REGION Network 42: Assign PLC Alarm Text List
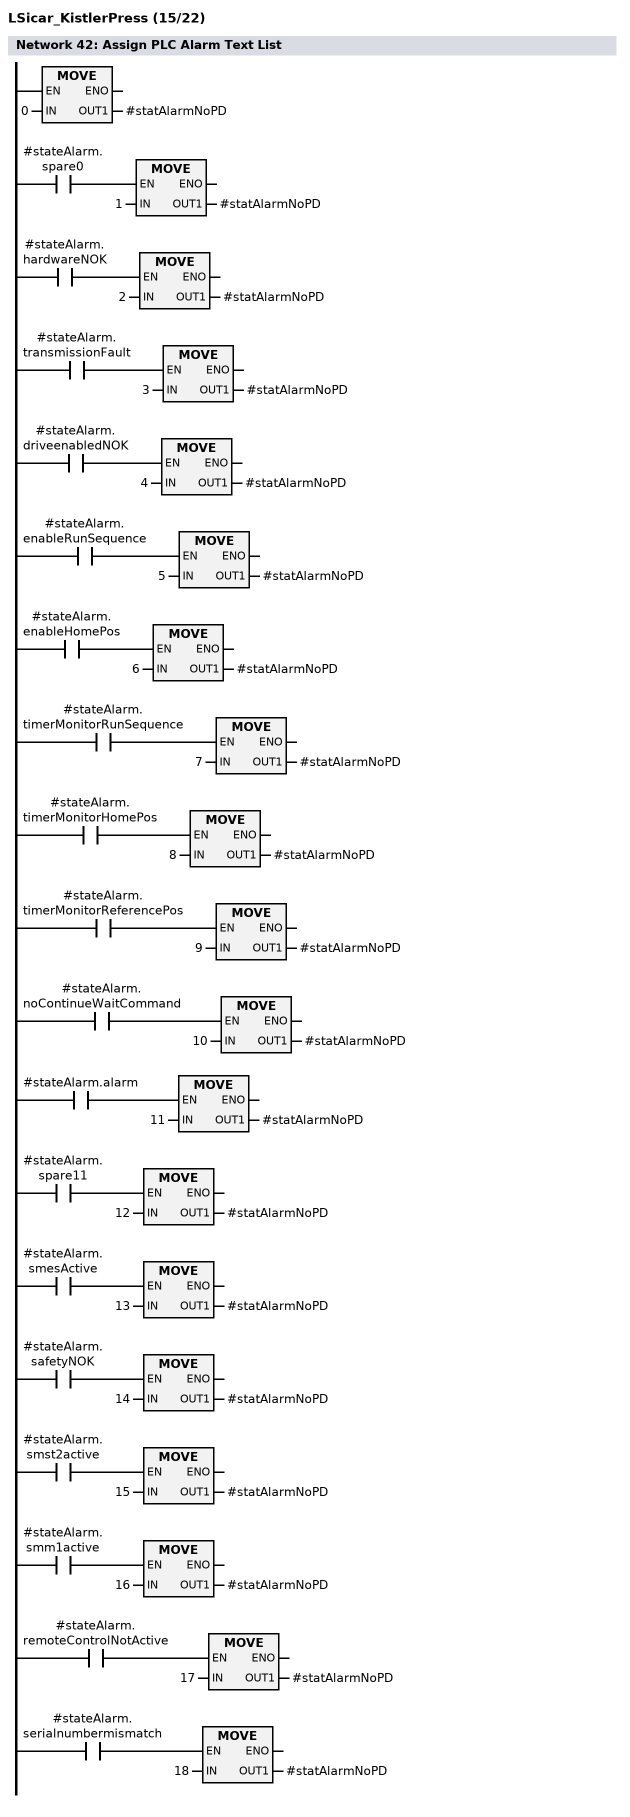
   RUNG wire#powerrail
      Move(in := 0, out1 => #statAlarmNoPD)
   END_RUNG
   RUNG wire#powerrail
      Contact( #stateAlarm.spare0 )
      Move(in := 1, out1 => #statAlarmNoPD)
   END_RUNG
   RUNG wire#powerrail
      Contact( #stateAlarm.hardwareNOK )
      Move(in := 2, out1 => #statAlarmNoPD)
   END_RUNG
   RUNG wire#powerrail
      Contact( #stateAlarm.transmissionFault )
      Move(in := 3, out1 => #statAlarmNoPD)
   END_RUNG
   RUNG wire#powerrail
      Contact( #stateAlarm.driveenabledNOK )
      Move(in := 4, out1 => #statAlarmNoPD)
   END_RUNG
   RUNG wire#powerrail
      Contact( #stateAlarm.enableRunSequence )
      Move(in := 5, out1 => #statAlarmNoPD)
   END_RUNG
   RUNG wire#powerrail
      Contact( #stateAlarm.enableHomePos )
      Move(in := 6, out1 => #statAlarmNoPD)
   END_RUNG
   RUNG wire#powerrail
      Contact( #stateAlarm.timerMonitorRunSequence )
      Move(in := 7, out1 => #statAlarmNoPD)
   END_RUNG
   RUNG wire#powerrail
      Contact( #stateAlarm.timerMonitorHomePos )
      Move(in := 8, out1 => #statAlarmNoPD)
   END_RUNG
   RUNG wire#powerrail
      Contact( #stateAlarm.timerMonitorReferencePos )
      Move(in := 9, out1 => #statAlarmNoPD)
   END_RUNG
   RUNG wire#powerrail
      Contact( #stateAlarm.noContinueWaitCommand )
      Move(in := 10, out1 => #statAlarmNoPD)
   END_RUNG
   RUNG wire#powerrail
      Contact( #stateAlarm.alarm )
      Move(in := 11, out1 => #statAlarmNoPD)
   END_RUNG
   RUNG wire#powerrail
      Contact( #stateAlarm.spare11 )
      Move(in := 12, out1 => #statAlarmNoPD)
   END_RUNG
   RUNG wire#powerrail
      Contact( #stateAlarm.smesActive )
      Move(in := 13, out1 => #statAlarmNoPD)
   END_RUNG
   RUNG wire#powerrail
      Contact( #stateAlarm.safetyNOK )
      Move(in := 14, out1 => #statAlarmNoPD)
   END_RUNG
   RUNG wire#powerrail
      Contact( #stateAlarm.smst2active )
      Move(in := 15, out1 => #statAlarmNoPD)
   END_RUNG
   RUNG wire#powerrail
      Contact( #stateAlarm.smm1active )
      Move(in := 16, out1 => #statAlarmNoPD)
   END_RUNG
   RUNG wire#powerrail
      Contact( #stateAlarm.remoteControlNotActive )
      Move(in := 17, out1 => #statAlarmNoPD)
   END_RUNG
   RUNG wire#powerrail
      Contact( #stateAlarm.serialnumbermismatch )
      Move(in := 18, out1 => #statAlarmNoPD)
   END_RUNG
   // the same network as SCL:
   #statAlarmNoPD := 0;
   IF #stateAlarm.spare0 THEN #statAlarmNoPD := 1; END_IF;
   IF #stateAlarm.hardwareNOK THEN #statAlarmNoPD := 2; END_IF;
   IF #stateAlarm.transmissionFault THEN #statAlarmNoPD := 3; END_IF;
   IF #stateAlarm.driveenabledNOK THEN #statAlarmNoPD := 4; END_IF;
   IF #stateAlarm.enableRunSequence THEN #statAlarmNoPD := 5; END_IF;
   IF #stateAlarm.enableHomePos THEN #statAlarmNoPD := 6; END_IF;
   IF #stateAlarm.timerMonitorRunSequence THEN #statAlarmNoPD := 7; END_IF;
   IF #stateAlarm.timerMonitorHomePos THEN #statAlarmNoPD := 8; END_IF;
   IF #stateAlarm.timerMonitorReferencePos THEN #statAlarmNoPD := 9; END_IF;
   IF #stateAlarm.noContinueWaitCommand THEN #statAlarmNoPD := 10; END_IF;
   IF #stateAlarm.alarm THEN #statAlarmNoPD := 11; END_IF;
   IF #stateAlarm.spare11 THEN #statAlarmNoPD := 12; END_IF;
   IF #stateAlarm.smesActive THEN #statAlarmNoPD := 13; END_IF;
   IF #stateAlarm.safetyNOK THEN #statAlarmNoPD := 14; END_IF;
   IF #stateAlarm.smst2active THEN #statAlarmNoPD := 15; END_IF;
   IF #stateAlarm.smm1active THEN #statAlarmNoPD := 16; END_IF;
   IF #stateAlarm.remoteControlNotActive THEN #statAlarmNoPD := 17; END_IF;
   IF #stateAlarm.serialnumbermismatch THEN #statAlarmNoPD := 18; END_IF;
END_REGION

REGION Network 43: HMI Color Association
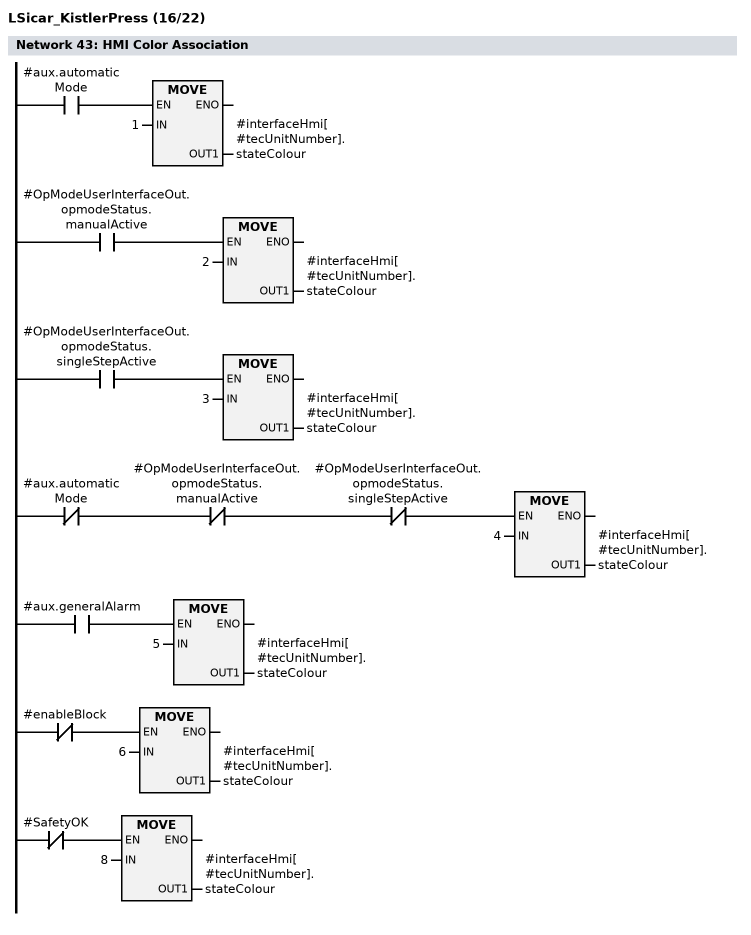
   RUNG wire#powerrail
      Contact( #aux.automaticMode )
      Move(in := 1, out1 => #interfaceHmi[#tecUnitNumber].stateColour)
   END_RUNG
   RUNG wire#powerrail
      Contact( #OpModeUserInterfaceOut.opmodeStatus.manualActive )
      Move(in := 2, out1 => #interfaceHmi[#tecUnitNumber].stateColour)
   END_RUNG
   RUNG wire#powerrail
      Contact( #OpModeUserInterfaceOut.opmodeStatus.singleStepActive )
      Move(in := 3, out1 => #interfaceHmi[#tecUnitNumber].stateColour)
   END_RUNG
   RUNG wire#powerrail
      I_Contact( #aux.automaticMode )
      I_Contact( #OpModeUserInterfaceOut.opmodeStatus.manualActive )
      I_Contact( #OpModeUserInterfaceOut.opmodeStatus.singleStepActive )
      Move(in := 4, out1 => #interfaceHmi[#tecUnitNumber].stateColour)
   END_RUNG
   RUNG wire#powerrail
      Contact( #aux.generalAlarm )
      Move(in := 5, out1 => #interfaceHmi[#tecUnitNumber].stateColour)
   END_RUNG
   RUNG wire#powerrail
      I_Contact( #enableBlock )
      Move(in := 6, out1 => #interfaceHmi[#tecUnitNumber].stateColour)
   END_RUNG
   RUNG wire#powerrail
      I_Contact( #SafetyOK )
      Move(in := 8, out1 => #interfaceHmi[#tecUnitNumber].stateColour)
   END_RUNG
   // the same network as SCL:
   IF #aux.automaticMode THEN #interfaceHmi[#tecUnitNumber].stateColour := 1; END_IF;
   IF #OpModeUserInterfaceOut.opmodeStatus.manualActive THEN
       #interfaceHmi[#tecUnitNumber].stateColour := 2;
   END_IF;
   IF #OpModeUserInterfaceOut.opmodeStatus.singleStepActive THEN
       #interfaceHmi[#tecUnitNumber].stateColour := 3;
   END_IF;
   IF NOT #aux.automaticMode AND NOT #OpModeUserInterfaceOut.opmodeStatus.manualActive AND NOT #OpModeUserInterfaceOut.opmodeStatus.singleStepActive THEN
       #interfaceHmi[#tecUnitNumber].stateColour := 4;
   END_IF;
   IF #aux.generalAlarm THEN #interfaceHmi[#tecUnitNumber].stateColour := 5; END_IF;
   IF NOT #enableBlock THEN #interfaceHmi[#tecUnitNumber].stateColour := 6; END_IF;
   IF NOT #SafetyOK THEN #interfaceHmi[#tecUnitNumber].stateColour := 8; END_IF;
END_REGION

REGION Network 44: HMI state Mapping
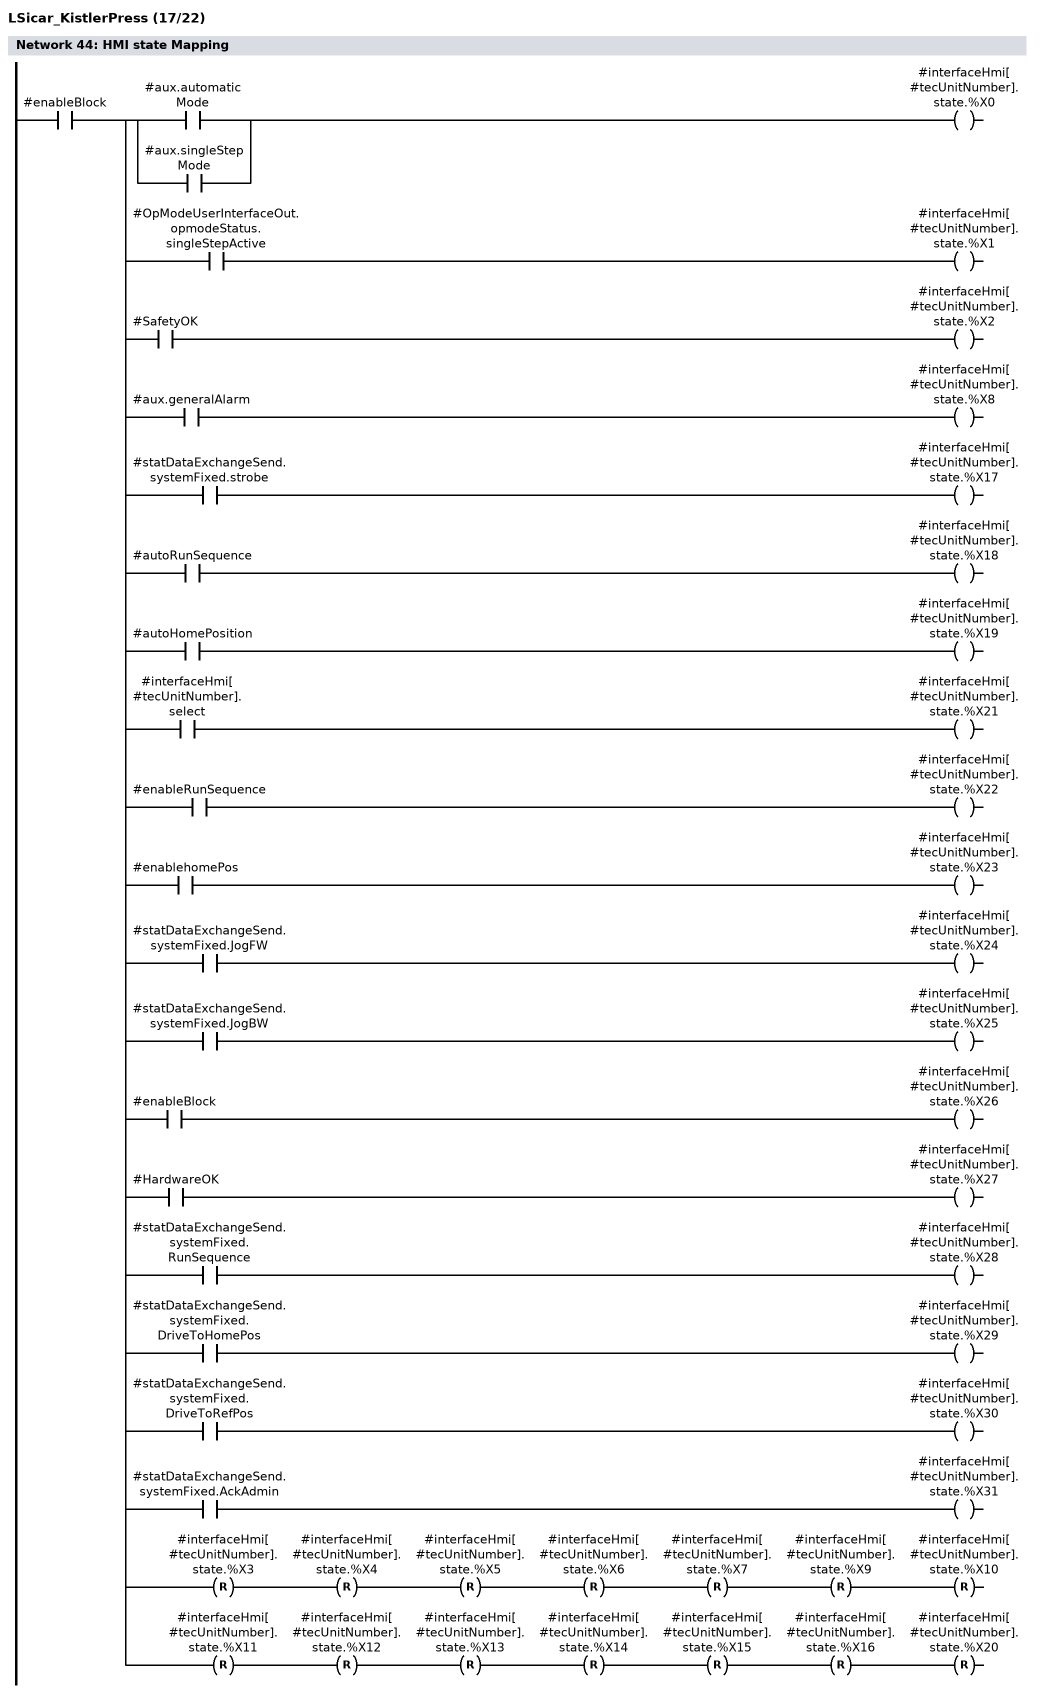
   RUNG wire#powerrail
      Contact( #enableBlock )
      wire#w1
      Contact( #aux.automaticMode )
      wire#w2
      Coil( #interfaceHmi[#tecUnitNumber].state.%X0 )
   END_RUNG
   RUNG wire#w1
      Contact( #aux.singleStepMode )
   END_RUNG wire#w2
   RUNG wire#w1
      Contact( #OpModeUserInterfaceOut.opmodeStatus.singleStepActive )
      Coil( #interfaceHmi[#tecUnitNumber].state.%X1 )
   END_RUNG
   RUNG wire#w1
      Contact( #SafetyOK )
      Coil( #interfaceHmi[#tecUnitNumber].state.%X2 )
   END_RUNG
   RUNG wire#w1
      Contact( #aux.generalAlarm )
      Coil( #interfaceHmi[#tecUnitNumber].state.%X8 )
   END_RUNG
   RUNG wire#w1
      Contact( #statDataExchangeSend.systemFixed.strobe )
      Coil( #interfaceHmi[#tecUnitNumber].state.%X17 )
   END_RUNG
   RUNG wire#w1
      Contact( #autoRunSequence )
      Coil( #interfaceHmi[#tecUnitNumber].state.%X18 )
   END_RUNG
   RUNG wire#w1
      Contact( #autoHomePosition )
      Coil( #interfaceHmi[#tecUnitNumber].state.%X19 )
   END_RUNG
   RUNG wire#w1
      Contact( #interfaceHmi[#tecUnitNumber].select )
      Coil( #interfaceHmi[#tecUnitNumber].state.%X21 )
   END_RUNG
   RUNG wire#w1
      Contact( #enableRunSequence )
      Coil( #interfaceHmi[#tecUnitNumber].state.%X22 )
   END_RUNG
   RUNG wire#w1
      Contact( #enablehomePos )
      Coil( #interfaceHmi[#tecUnitNumber].state.%X23 )
   END_RUNG
   RUNG wire#w1
      Contact( #statDataExchangeSend.systemFixed.JogFW )
      Coil( #interfaceHmi[#tecUnitNumber].state.%X24 )
   END_RUNG
   RUNG wire#w1
      Contact( #statDataExchangeSend.systemFixed.JogBW )
      Coil( #interfaceHmi[#tecUnitNumber].state.%X25 )
   END_RUNG
   RUNG wire#w1
      Contact( #enableBlock )
      Coil( #interfaceHmi[#tecUnitNumber].state.%X26 )
   END_RUNG
   RUNG wire#w1
      Contact( #HardwareOK )
      Coil( #interfaceHmi[#tecUnitNumber].state.%X27 )
   END_RUNG
   RUNG wire#w1
      Contact( #statDataExchangeSend.systemFixed.RunSequence )
      Coil( #interfaceHmi[#tecUnitNumber].state.%X28 )
   END_RUNG
   RUNG wire#w1
      Contact( #statDataExchangeSend.systemFixed.DriveToHomePos )
      Coil( #interfaceHmi[#tecUnitNumber].state.%X29 )
   END_RUNG
   RUNG wire#w1
      Contact( #statDataExchangeSend.systemFixed.DriveToRefPos )
      Coil( #interfaceHmi[#tecUnitNumber].state.%X30 )
   END_RUNG
   RUNG wire#w1
      Contact( #statDataExchangeSend.systemFixed.AckAdmin )
      Coil( #interfaceHmi[#tecUnitNumber].state.%X31 )
   END_RUNG
   RUNG wire#w1
      R_Coil( #interfaceHmi[#tecUnitNumber].state.%X3 )
      R_Coil( #interfaceHmi[#tecUnitNumber].state.%X4 )
      R_Coil( #interfaceHmi[#tecUnitNumber].state.%X5 )
      R_Coil( #interfaceHmi[#tecUnitNumber].state.%X6 )
      R_Coil( #interfaceHmi[#tecUnitNumber].state.%X7 )
      R_Coil( #interfaceHmi[#tecUnitNumber].state.%X9 )
      R_Coil( #interfaceHmi[#tecUnitNumber].state.%X10 )
   END_RUNG
   RUNG wire#w1
      R_Coil( #interfaceHmi[#tecUnitNumber].state.%X11 )
      R_Coil( #interfaceHmi[#tecUnitNumber].state.%X12 )
      R_Coil( #interfaceHmi[#tecUnitNumber].state.%X13 )
      R_Coil( #interfaceHmi[#tecUnitNumber].state.%X14 )
      R_Coil( #interfaceHmi[#tecUnitNumber].state.%X15 )
      R_Coil( #interfaceHmi[#tecUnitNumber].state.%X16 )
      R_Coil( #interfaceHmi[#tecUnitNumber].state.%X20 )
   END_RUNG
   // the same network as SCL:
   #interfaceHmi[#tecUnitNumber].state.%X0 := #enableBlock AND (#aux.automaticMode OR #aux.singleStepMode);
   #interfaceHmi[#tecUnitNumber].state.%X1 := #enableBlock AND #OpModeUserInterfaceOut.opmodeStatus.singleStepActive;
   #interfaceHmi[#tecUnitNumber].state.%X2 := #enableBlock AND #SafetyOK;
   #interfaceHmi[#tecUnitNumber].state.%X8 := #enableBlock AND #aux.generalAlarm;
   #interfaceHmi[#tecUnitNumber].state.%X17 := #enableBlock AND #statDataExchangeSend.systemFixed.strobe;
   #interfaceHmi[#tecUnitNumber].state.%X18 := #enableBlock AND #autoRunSequence;
   #interfaceHmi[#tecUnitNumber].state.%X19 := #enableBlock AND #autoHomePosition;
   #interfaceHmi[#tecUnitNumber].state.%X21 := #enableBlock AND #interfaceHmi[#tecUnitNumber].select;
   #interfaceHmi[#tecUnitNumber].state.%X22 := #enableBlock AND #enableRunSequence;
   #interfaceHmi[#tecUnitNumber].state.%X23 := #enableBlock AND #enablehomePos;
   #interfaceHmi[#tecUnitNumber].state.%X24 := #enableBlock AND #statDataExchangeSend.systemFixed.JogFW;
   #interfaceHmi[#tecUnitNumber].state.%X25 := #enableBlock AND #statDataExchangeSend.systemFixed.JogBW;
   #interfaceHmi[#tecUnitNumber].state.%X26 := #enableBlock AND #enableBlock;
   #interfaceHmi[#tecUnitNumber].state.%X27 := #enableBlock AND #HardwareOK;
   #interfaceHmi[#tecUnitNumber].state.%X28 := #enableBlock AND #statDataExchangeSend.systemFixed.RunSequence;
   #interfaceHmi[#tecUnitNumber].state.%X29 := #enableBlock AND #statDataExchangeSend.systemFixed.DriveToHomePos;
   #interfaceHmi[#tecUnitNumber].state.%X30 := #enableBlock AND #statDataExchangeSend.systemFixed.DriveToRefPos;
   #interfaceHmi[#tecUnitNumber].state.%X31 := #enableBlock AND #statDataExchangeSend.systemFixed.AckAdmin;
   IF #enableBlock THEN
       #interfaceHmi[#tecUnitNumber].state.%X3 := FALSE;
       #interfaceHmi[#tecUnitNumber].state.%X4 := FALSE;
       #interfaceHmi[#tecUnitNumber].state.%X5 := FALSE;
       #interfaceHmi[#tecUnitNumber].state.%X6 := FALSE;
       #interfaceHmi[#tecUnitNumber].state.%X7 := FALSE;
       #interfaceHmi[#tecUnitNumber].state.%X9 := FALSE;
       #interfaceHmi[#tecUnitNumber].state.%X10 := FALSE;
       #interfaceHmi[#tecUnitNumber].state.%X11 := FALSE;
       #interfaceHmi[#tecUnitNumber].state.%X12 := FALSE;
       #interfaceHmi[#tecUnitNumber].state.%X13 := FALSE;
       #interfaceHmi[#tecUnitNumber].state.%X14 := FALSE;
       #interfaceHmi[#tecUnitNumber].state.%X15 := FALSE;
       #interfaceHmi[#tecUnitNumber].state.%X16 := FALSE;
       #interfaceHmi[#tecUnitNumber].state.%X20 := FALSE;
   END_IF;
END_REGION

REGION Network 45: Send Process Values to HMI
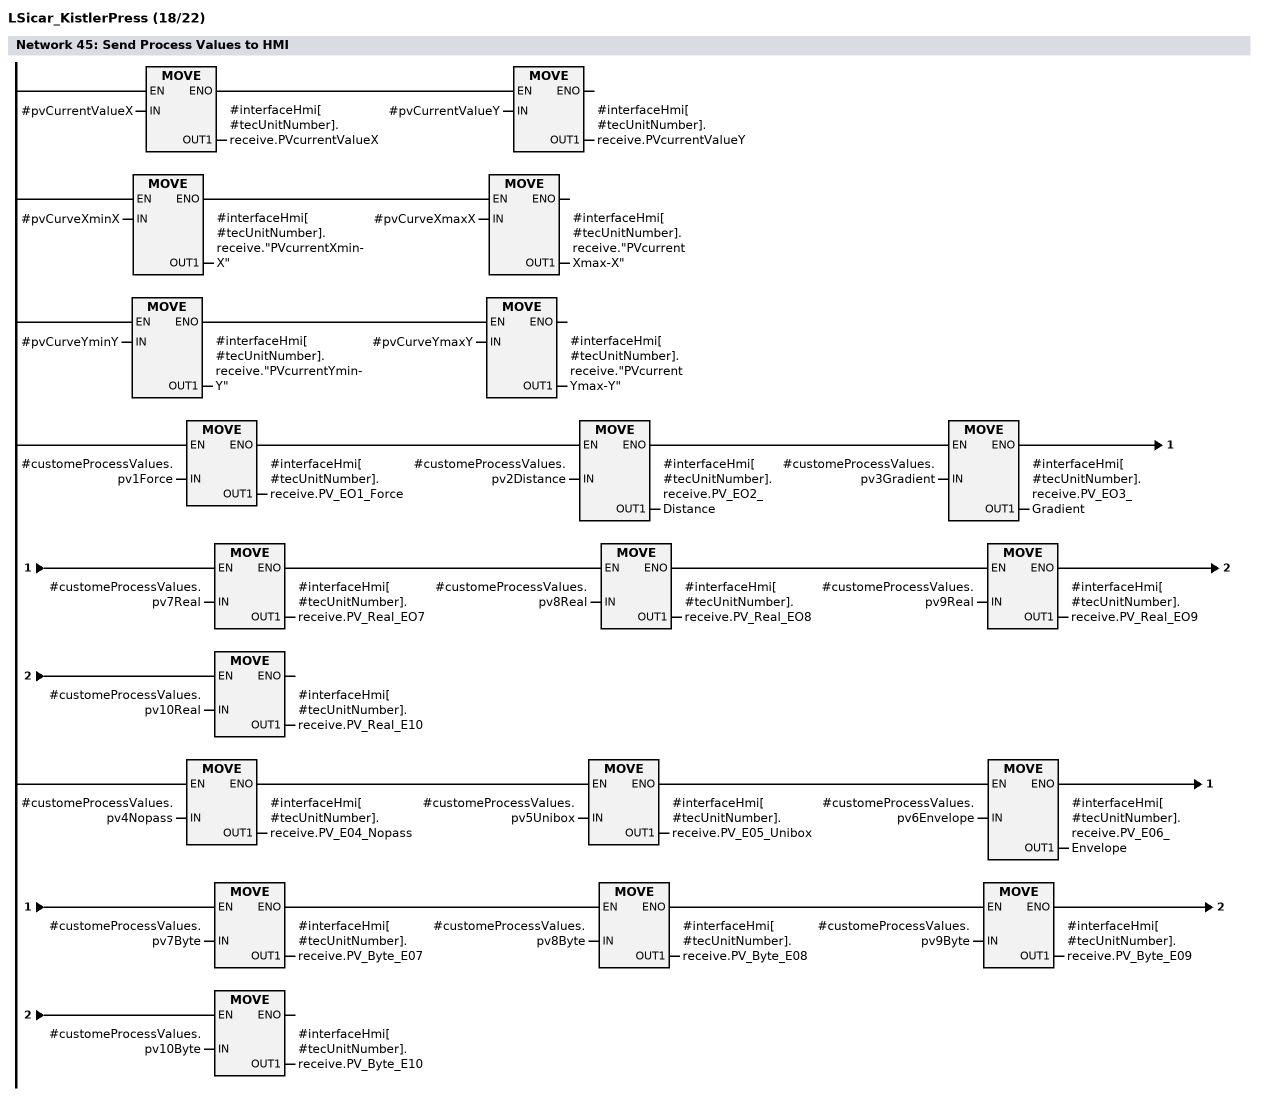
   RUNG wire#powerrail
      Move(in := #pvCurrentValueX, out1 => #interfaceHmi[#tecUnitNumber].receive.PVcurrentValueX)
      Move(in := #pvCurrentValueY, out1 => #interfaceHmi[#tecUnitNumber].receive.PVcurrentValueY)
   END_RUNG
   RUNG wire#powerrail
      Move(in := #pvCurveXminX, out1 => #interfaceHmi[#tecUnitNumber].receive."PVcurrentXmin-X")
      Move(in := #pvCurveXmaxX, out1 => #interfaceHmi[#tecUnitNumber].receive."PVcurrentXmax-X")
   END_RUNG
   RUNG wire#powerrail
      Move(in := #pvCurveYminY, out1 => #interfaceHmi[#tecUnitNumber].receive."PVcurrentYmin-Y")
      Move(in := #pvCurveYmaxY, out1 => #interfaceHmi[#tecUnitNumber].receive."PVcurrentYmax-Y")
   END_RUNG
   RUNG wire#powerrail
      Move(in := #customeProcessValues.pv1Force, out1 => #interfaceHmi[#tecUnitNumber].receive.PV_EO1_Force)
      Move(in := #customeProcessValues.pv2Distance, out1 => #interfaceHmi[#tecUnitNumber].receive.PV_EO2_Distance)
      Move(in := #customeProcessValues.pv3Gradient, out1 => #interfaceHmi[#tecUnitNumber].receive.PV_EO3_Gradient)
      Move(in := #customeProcessValues.pv7Real, out1 => #interfaceHmi[#tecUnitNumber].receive.PV_Real_EO7)
      Move(in := #customeProcessValues.pv8Real, out1 => #interfaceHmi[#tecUnitNumber].receive.PV_Real_EO8)
      Move(in := #customeProcessValues.pv9Real, out1 => #interfaceHmi[#tecUnitNumber].receive.PV_Real_EO9)
      Move(in := #customeProcessValues.pv10Real, out1 => #interfaceHmi[#tecUnitNumber].receive.PV_Real_E10)
   END_RUNG
   RUNG wire#powerrail
      Move(in := #customeProcessValues.pv4Nopass, out1 => #interfaceHmi[#tecUnitNumber].receive.PV_E04_Nopass)
      Move(in := #customeProcessValues.pv5Unibox, out1 => #interfaceHmi[#tecUnitNumber].receive.PV_E05_Unibox)
      Move(in := #customeProcessValues.pv6Envelope, out1 => #interfaceHmi[#tecUnitNumber].receive.PV_E06_Envelope)
      Move(in := #customeProcessValues.pv7Byte, out1 => #interfaceHmi[#tecUnitNumber].receive.PV_Byte_E07)
      Move(in := #customeProcessValues.pv8Byte, out1 => #interfaceHmi[#tecUnitNumber].receive.PV_Byte_E08)
      Move(in := #customeProcessValues.pv9Byte, out1 => #interfaceHmi[#tecUnitNumber].receive.PV_Byte_E09)
      Move(in := #customeProcessValues.pv10Byte, out1 => #interfaceHmi[#tecUnitNumber].receive.PV_Byte_E10)
   END_RUNG
   // the same network as SCL:
   #interfaceHmi[#tecUnitNumber].receive.PVcurrentValueX := #pvCurrentValueX;
   #interfaceHmi[#tecUnitNumber].receive.PVcurrentValueY := #pvCurrentValueY;
   #interfaceHmi[#tecUnitNumber].receive."PVcurrentXmin-X" := #pvCurveXminX;
   #interfaceHmi[#tecUnitNumber].receive."PVcurrentXmax-X" := #pvCurveXmaxX;
   #interfaceHmi[#tecUnitNumber].receive."PVcurrentYmin-Y" := #pvCurveYminY;
   #interfaceHmi[#tecUnitNumber].receive."PVcurrentYmax-Y" := #pvCurveYmaxY;
   #interfaceHmi[#tecUnitNumber].receive.PV_EO1_Force := #customeProcessValues.pv1Force;
   #interfaceHmi[#tecUnitNumber].receive.PV_EO2_Distance := #customeProcessValues.pv2Distance;
   #interfaceHmi[#tecUnitNumber].receive.PV_EO3_Gradient := #customeProcessValues.pv3Gradient;
   #interfaceHmi[#tecUnitNumber].receive.PV_Real_EO7 := #customeProcessValues.pv7Real;
   #interfaceHmi[#tecUnitNumber].receive.PV_Real_EO8 := #customeProcessValues.pv8Real;
   #interfaceHmi[#tecUnitNumber].receive.PV_Real_EO9 := #customeProcessValues.pv9Real;
   #interfaceHmi[#tecUnitNumber].receive.PV_Real_E10 := #customeProcessValues.pv10Real;
   #interfaceHmi[#tecUnitNumber].receive.PV_E04_Nopass := #customeProcessValues.pv4Nopass;
   #interfaceHmi[#tecUnitNumber].receive.PV_E05_Unibox := #customeProcessValues.pv5Unibox;
   #interfaceHmi[#tecUnitNumber].receive.PV_E06_Envelope := #customeProcessValues.pv6Envelope;
   #interfaceHmi[#tecUnitNumber].receive.PV_Byte_E07 := #customeProcessValues.pv7Byte;
   #interfaceHmi[#tecUnitNumber].receive.PV_Byte_E08 := #customeProcessValues.pv8Byte;
   #interfaceHmi[#tecUnitNumber].receive.PV_Byte_E09 := #customeProcessValues.pv9Byte;
   #interfaceHmi[#tecUnitNumber].receive.PV_Byte_E10 := #customeProcessValues.pv10Byte;
END_REGION

REGION Network 46: Enable HMI Code View
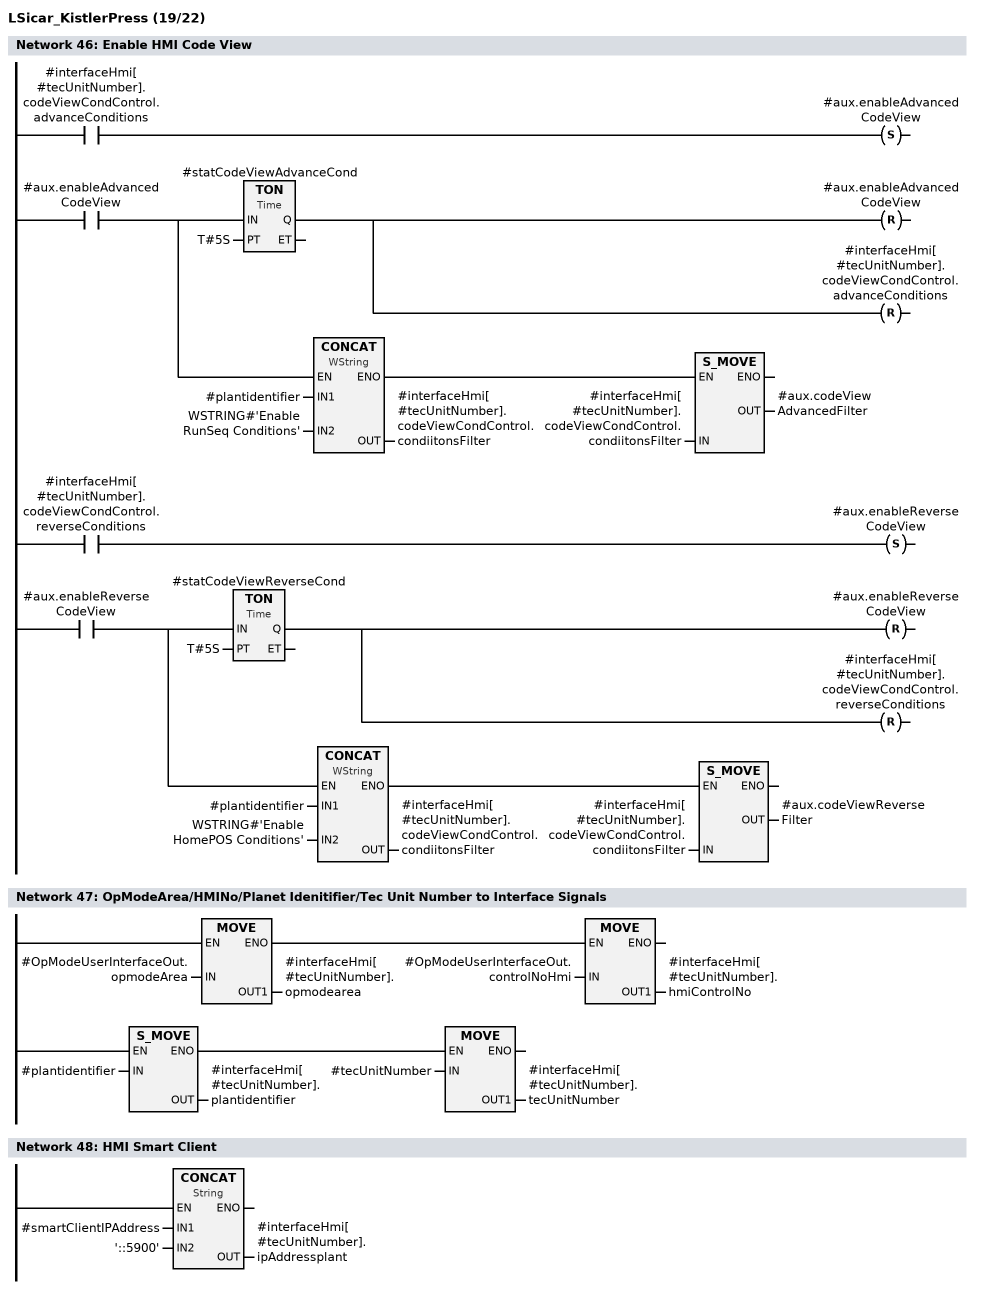
   RUNG wire#powerrail
      Contact( #interfaceHmi[#tecUnitNumber].codeViewCondControl.advanceConditions )
      S_Coil( #aux.enableAdvancedCodeView )
   END_RUNG
   RUNG wire#powerrail
      Contact( #aux.enableAdvancedCodeView )
      wire#w1
      { S7_Templates := "time_type := Time" } #statCodeViewAdvanceCond.TON(pt := T#5S, et =>)
      wire#w2
      R_Coil( #aux.enableAdvancedCodeView )
   END_RUNG
   RUNG wire#w2
      R_Coil( #interfaceHmi[#tecUnitNumber].codeViewCondControl.advanceConditions )
   END_RUNG
   RUNG wire#w1
      { S7_Templates := "[card := 2, str_type := WString]" } CONCAT(IN1 := #plantidentifier, IN2 := WSTRING#'Enable RunSeq Conditions', OUT => #interfaceHmi[#tecUnitNumber].codeViewCondControl.condiitonsFilter)
      S_Move(in := #interfaceHmi[#tecUnitNumber].codeViewCondControl.condiitonsFilter, out => #aux.codeViewAdvancedFilter)
   END_RUNG
   RUNG wire#powerrail
      Contact( #interfaceHmi[#tecUnitNumber].codeViewCondControl.reverseConditions )
      S_Coil( #aux.enableReverseCodeView )
   END_RUNG
   RUNG wire#powerrail
      Contact( #aux.enableReverseCodeView )
      wire#w3
      { S7_Templates := "time_type := Time" } #statCodeViewReverseCond.TON(pt := T#5S, et =>)
      wire#w4
      R_Coil( #aux.enableReverseCodeView )
   END_RUNG
   RUNG wire#w4
      R_Coil( #interfaceHmi[#tecUnitNumber].codeViewCondControl.reverseConditions )
   END_RUNG
   RUNG wire#w3
      { S7_Templates := "[card := 2, str_type := WString]" } CONCAT(IN1 := #plantidentifier, IN2 := WSTRING#'Enable HomePOS Conditions', OUT => #interfaceHmi[#tecUnitNumber].codeViewCondControl.condiitonsFilter)
      S_Move(in := #interfaceHmi[#tecUnitNumber].codeViewCondControl.condiitonsFilter, out => #aux.codeViewReverseFilter)
   END_RUNG
   // the same network as SCL:
   IF #interfaceHmi[#tecUnitNumber].codeViewCondControl.advanceConditions THEN
       #aux.enableAdvancedCodeView := TRUE;
   END_IF;
   #statCodeViewAdvanceCond(IN := #aux.enableAdvancedCodeView, PT := T#5S);   // TON
   #_w1 := #aux.enableAdvancedCodeView;
   IF #statCodeViewAdvanceCond.Q THEN
       #aux.enableAdvancedCodeView := FALSE;
       #interfaceHmi[#tecUnitNumber].codeViewCondControl.advanceConditions := FALSE;
   END_IF;
   CONCAT(EN := #_w1,
          IN1 := #plantidentifier,
          IN2 := WSTRING#'Enable RunSeq Conditions',
          OUT => #interfaceHmi[#tecUnitNumber].codeViewCondControl.condiitonsFilter,
          ENO => #_w2);
   IF #_w2 THEN
       #aux.codeViewAdvancedFilter := #interfaceHmi[#tecUnitNumber].codeViewCondControl.condiitonsFilter;
   END_IF;
   IF #interfaceHmi[#tecUnitNumber].codeViewCondControl.reverseConditions THEN
       #aux.enableReverseCodeView := TRUE;
   END_IF;
   #statCodeViewReverseCond(IN := #aux.enableReverseCodeView, PT := T#5S);   // TON
   #_w3 := #aux.enableReverseCodeView;
   IF #statCodeViewReverseCond.Q THEN
       #aux.enableReverseCodeView := FALSE;
       #interfaceHmi[#tecUnitNumber].codeViewCondControl.reverseConditions := FALSE;
   END_IF;
   CONCAT(EN := #_w3,
          IN1 := #plantidentifier,
          IN2 := WSTRING#'Enable HomePOS Conditions',
          OUT => #interfaceHmi[#tecUnitNumber].codeViewCondControl.condiitonsFilter,
          ENO => #_w4);
   IF #_w4 THEN
       #aux.codeViewReverseFilter := #interfaceHmi[#tecUnitNumber].codeViewCondControl.condiitonsFilter;
   END_IF;
END_REGION

REGION Network 47: OpModeArea/HMINo/Planet Idenitifier/Tec Unit Number to Interface Signals
   RUNG wire#powerrail
      Move(in := #OpModeUserInterfaceOut.opmodeArea, out1 => #interfaceHmi[#tecUnitNumber].opmodearea)
      Move(in := #OpModeUserInterfaceOut.controlNoHmi, out1 => #interfaceHmi[#tecUnitNumber].hmiControlNo)
   END_RUNG
   RUNG wire#powerrail
      S_Move(in := #plantidentifier, out => #interfaceHmi[#tecUnitNumber].plantidentifier)
      Move(in := #tecUnitNumber, out1 => #interfaceHmi[#tecUnitNumber].tecUnitNumber)
   END_RUNG
   // the same network as SCL:
   #interfaceHmi[#tecUnitNumber].opmodearea := #OpModeUserInterfaceOut.opmodeArea;
   #interfaceHmi[#tecUnitNumber].hmiControlNo := #OpModeUserInterfaceOut.controlNoHmi;
   #interfaceHmi[#tecUnitNumber].plantidentifier := #plantidentifier;
   #interfaceHmi[#tecUnitNumber].tecUnitNumber := #tecUnitNumber;
END_REGION

REGION Network 48: HMI Smart Client
   RUNG wire#powerrail
      { S7_Templates := "[card := 2, str_type := String]" } CONCAT(IN1 := #smartClientIPAddress, IN2 := '::5900', OUT => #interfaceHmi[#tecUnitNumber].ipAddressplant)
   END_RUNG
   // the same network as SCL:
   CONCAT(IN1 := #smartClientIPAddress, IN2 := '::5900', OUT => #interfaceHmi[#tecUnitNumber].ipAddressplant);
END_REGION

REGION Network 49: Map FIx Receieved Data to HMI
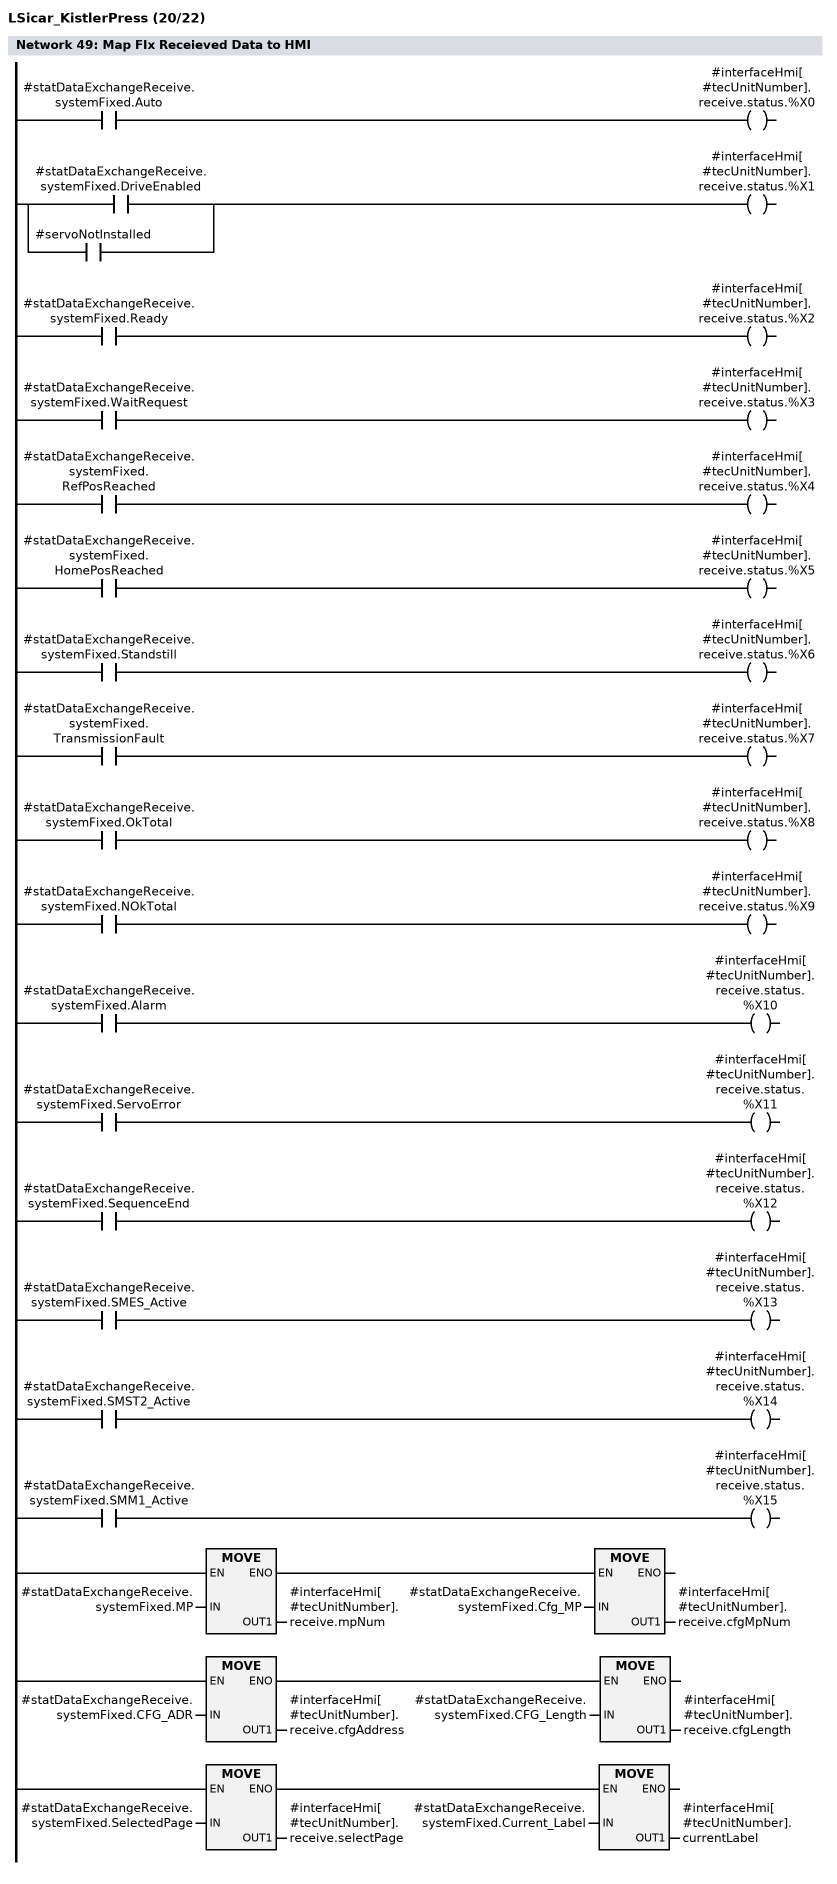
   RUNG wire#powerrail
      Contact( #statDataExchangeReceive.systemFixed.Auto )
      Coil( #interfaceHmi[#tecUnitNumber].receive.status.%X0 )
   END_RUNG
   RUNG wire#powerrail
      Contact( #statDataExchangeReceive.systemFixed.DriveEnabled )
      wire#w1
      Coil( #interfaceHmi[#tecUnitNumber].receive.status.%X1 )
   END_RUNG
   RUNG wire#powerrail
      Contact( #servoNotInstalled )
   END_RUNG wire#w1
   RUNG wire#powerrail
      Contact( #statDataExchangeReceive.systemFixed.Ready )
      Coil( #interfaceHmi[#tecUnitNumber].receive.status.%X2 )
   END_RUNG
   RUNG wire#powerrail
      Contact( #statDataExchangeReceive.systemFixed.WaitRequest )
      Coil( #interfaceHmi[#tecUnitNumber].receive.status.%X3 )
   END_RUNG
   RUNG wire#powerrail
      Contact( #statDataExchangeReceive.systemFixed.RefPosReached )
      Coil( #interfaceHmi[#tecUnitNumber].receive.status.%X4 )
   END_RUNG
   RUNG wire#powerrail
      Contact( #statDataExchangeReceive.systemFixed.HomePosReached )
      Coil( #interfaceHmi[#tecUnitNumber].receive.status.%X5 )
   END_RUNG
   RUNG wire#powerrail
      Contact( #statDataExchangeReceive.systemFixed.Standstill )
      Coil( #interfaceHmi[#tecUnitNumber].receive.status.%X6 )
   END_RUNG
   RUNG wire#powerrail
      Contact( #statDataExchangeReceive.systemFixed.TransmissionFault )
      Coil( #interfaceHmi[#tecUnitNumber].receive.status.%X7 )
   END_RUNG
   RUNG wire#powerrail
      Contact( #statDataExchangeReceive.systemFixed.OkTotal )
      Coil( #interfaceHmi[#tecUnitNumber].receive.status.%X8 )
   END_RUNG
   RUNG wire#powerrail
      Contact( #statDataExchangeReceive.systemFixed.NOkTotal )
      Coil( #interfaceHmi[#tecUnitNumber].receive.status.%X9 )
   END_RUNG
   RUNG wire#powerrail
      Contact( #statDataExchangeReceive.systemFixed.Alarm )
      Coil( #interfaceHmi[#tecUnitNumber].receive.status.%X10 )
   END_RUNG
   RUNG wire#powerrail
      Contact( #statDataExchangeReceive.systemFixed.ServoError )
      Coil( #interfaceHmi[#tecUnitNumber].receive.status.%X11 )
   END_RUNG
   RUNG wire#powerrail
      Contact( #statDataExchangeReceive.systemFixed.SequenceEnd )
      Coil( #interfaceHmi[#tecUnitNumber].receive.status.%X12 )
   END_RUNG
   RUNG wire#powerrail
      Contact( #statDataExchangeReceive.systemFixed.SMES_Active )
      Coil( #interfaceHmi[#tecUnitNumber].receive.status.%X13 )
   END_RUNG
   RUNG wire#powerrail
      Contact( #statDataExchangeReceive.systemFixed.SMST2_Active )
      Coil( #interfaceHmi[#tecUnitNumber].receive.status.%X14 )
   END_RUNG
   RUNG wire#powerrail
      Contact( #statDataExchangeReceive.systemFixed.SMM1_Active )
      Coil( #interfaceHmi[#tecUnitNumber].receive.status.%X15 )
   END_RUNG
   RUNG wire#powerrail
      Move(in := #statDataExchangeReceive.systemFixed.MP, out1 => #interfaceHmi[#tecUnitNumber].receive.mpNum)
      Move(in := #statDataExchangeReceive.systemFixed.Cfg_MP, out1 => #interfaceHmi[#tecUnitNumber].receive.cfgMpNum)
   END_RUNG
   RUNG wire#powerrail
      Move(in := #statDataExchangeReceive.systemFixed.CFG_ADR, out1 => #interfaceHmi[#tecUnitNumber].receive.cfgAddress)
      Move(in := #statDataExchangeReceive.systemFixed.CFG_Length, out1 => #interfaceHmi[#tecUnitNumber].receive.cfgLength)
   END_RUNG
   RUNG wire#powerrail
      Move(in := #statDataExchangeReceive.systemFixed.SelectedPage, out1 => #interfaceHmi[#tecUnitNumber].receive.selectPage)
      Move(in := #statDataExchangeReceive.systemFixed.Current_Label, out1 => #interfaceHmi[#tecUnitNumber].currentLabel)
   END_RUNG
   // the same network as SCL:
   #interfaceHmi[#tecUnitNumber].receive.status.%X0 := #statDataExchangeReceive.systemFixed.Auto;
   #interfaceHmi[#tecUnitNumber].receive.status.%X1 := #statDataExchangeReceive.systemFixed.DriveEnabled OR #servoNotInstalled;
   #interfaceHmi[#tecUnitNumber].receive.status.%X2 := #statDataExchangeReceive.systemFixed.Ready;
   #interfaceHmi[#tecUnitNumber].receive.status.%X3 := #statDataExchangeReceive.systemFixed.WaitRequest;
   #interfaceHmi[#tecUnitNumber].receive.status.%X4 := #statDataExchangeReceive.systemFixed.RefPosReached;
   #interfaceHmi[#tecUnitNumber].receive.status.%X5 := #statDataExchangeReceive.systemFixed.HomePosReached;
   #interfaceHmi[#tecUnitNumber].receive.status.%X6 := #statDataExchangeReceive.systemFixed.Standstill;
   #interfaceHmi[#tecUnitNumber].receive.status.%X7 := #statDataExchangeReceive.systemFixed.TransmissionFault;
   #interfaceHmi[#tecUnitNumber].receive.status.%X8 := #statDataExchangeReceive.systemFixed.OkTotal;
   #interfaceHmi[#tecUnitNumber].receive.status.%X9 := #statDataExchangeReceive.systemFixed.NOkTotal;
   #interfaceHmi[#tecUnitNumber].receive.status.%X10 := #statDataExchangeReceive.systemFixed.Alarm;
   #interfaceHmi[#tecUnitNumber].receive.status.%X11 := #statDataExchangeReceive.systemFixed.ServoError;
   #interfaceHmi[#tecUnitNumber].receive.status.%X12 := #statDataExchangeReceive.systemFixed.SequenceEnd;
   #interfaceHmi[#tecUnitNumber].receive.status.%X13 := #statDataExchangeReceive.systemFixed.SMES_Active;
   #interfaceHmi[#tecUnitNumber].receive.status.%X14 := #statDataExchangeReceive.systemFixed.SMST2_Active;
   #interfaceHmi[#tecUnitNumber].receive.status.%X15 := #statDataExchangeReceive.systemFixed.SMM1_Active;
   #interfaceHmi[#tecUnitNumber].receive.mpNum := #statDataExchangeReceive.systemFixed.MP;
   #interfaceHmi[#tecUnitNumber].receive.cfgMpNum := #statDataExchangeReceive.systemFixed.Cfg_MP;
   #interfaceHmi[#tecUnitNumber].receive.cfgAddress := #statDataExchangeReceive.systemFixed.CFG_ADR;
   #interfaceHmi[#tecUnitNumber].receive.cfgLength := #statDataExchangeReceive.systemFixed.CFG_Length;
   #interfaceHmi[#tecUnitNumber].receive.selectPage := #statDataExchangeReceive.systemFixed.SelectedPage;
   #interfaceHmi[#tecUnitNumber].currentLabel := #statDataExchangeReceive.systemFixed.Current_Label;
END_REGION

REGION Network 50: Map Fix Send Data to HMI
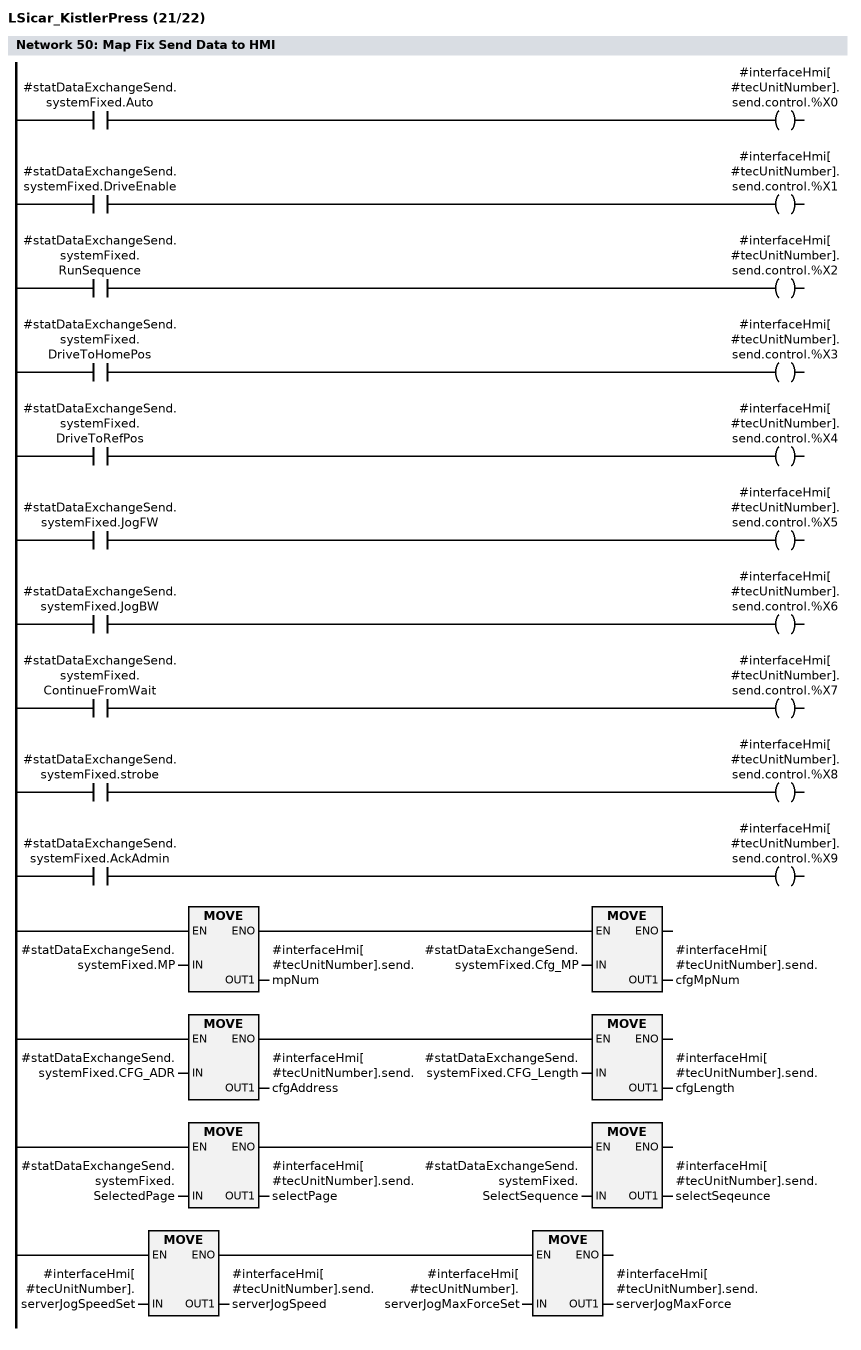
   RUNG wire#powerrail
      Contact( #statDataExchangeSend.systemFixed.Auto )
      Coil( #interfaceHmi[#tecUnitNumber].send.control.%X0 )
   END_RUNG
   RUNG wire#powerrail
      Contact( #statDataExchangeSend.systemFixed.DriveEnable )
      Coil( #interfaceHmi[#tecUnitNumber].send.control.%X1 )
   END_RUNG
   RUNG wire#powerrail
      Contact( #statDataExchangeSend.systemFixed.RunSequence )
      Coil( #interfaceHmi[#tecUnitNumber].send.control.%X2 )
   END_RUNG
   RUNG wire#powerrail
      Contact( #statDataExchangeSend.systemFixed.DriveToHomePos )
      Coil( #interfaceHmi[#tecUnitNumber].send.control.%X3 )
   END_RUNG
   RUNG wire#powerrail
      Contact( #statDataExchangeSend.systemFixed.DriveToRefPos )
      Coil( #interfaceHmi[#tecUnitNumber].send.control.%X4 )
   END_RUNG
   RUNG wire#powerrail
      Contact( #statDataExchangeSend.systemFixed.JogFW )
      Coil( #interfaceHmi[#tecUnitNumber].send.control.%X5 )
   END_RUNG
   RUNG wire#powerrail
      Contact( #statDataExchangeSend.systemFixed.JogBW )
      Coil( #interfaceHmi[#tecUnitNumber].send.control.%X6 )
   END_RUNG
   RUNG wire#powerrail
      Contact( #statDataExchangeSend.systemFixed.ContinueFromWait )
      Coil( #interfaceHmi[#tecUnitNumber].send.control.%X7 )
   END_RUNG
   RUNG wire#powerrail
      Contact( #statDataExchangeSend.systemFixed.strobe )
      Coil( #interfaceHmi[#tecUnitNumber].send.control.%X8 )
   END_RUNG
   RUNG wire#powerrail
      Contact( #statDataExchangeSend.systemFixed.AckAdmin )
      Coil( #interfaceHmi[#tecUnitNumber].send.control.%X9 )
   END_RUNG
   RUNG wire#powerrail
      Move(in := #statDataExchangeSend.systemFixed.MP, out1 => #interfaceHmi[#tecUnitNumber].send.mpNum)
      Move(in := #statDataExchangeSend.systemFixed.Cfg_MP, out1 => #interfaceHmi[#tecUnitNumber].send.cfgMpNum)
   END_RUNG
   RUNG wire#powerrail
      Move(in := #statDataExchangeSend.systemFixed.CFG_ADR, out1 => #interfaceHmi[#tecUnitNumber].send.cfgAddress)
      Move(in := #statDataExchangeSend.systemFixed.CFG_Length, out1 => #interfaceHmi[#tecUnitNumber].send.cfgLength)
   END_RUNG
   RUNG wire#powerrail
      Move(in := #statDataExchangeSend.systemFixed.SelectedPage, out1 => #interfaceHmi[#tecUnitNumber].send.selectPage)
      Move(in := #statDataExchangeSend.systemFixed.SelectSequence, out1 => #interfaceHmi[#tecUnitNumber].send.selectSeqeunce)
   END_RUNG
   RUNG wire#powerrail
      Move(in := #interfaceHmi[#tecUnitNumber].serverJogSpeedSet, out1 => #interfaceHmi[#tecUnitNumber].send.serverJogSpeed)
      Move(in := #interfaceHmi[#tecUnitNumber].serverJogMaxForceSet, out1 => #interfaceHmi[#tecUnitNumber].send.serverJogMaxForce)
   END_RUNG
   // the same network as SCL:
   #interfaceHmi[#tecUnitNumber].send.control.%X0 := #statDataExchangeSend.systemFixed.Auto;
   #interfaceHmi[#tecUnitNumber].send.control.%X1 := #statDataExchangeSend.systemFixed.DriveEnable;
   #interfaceHmi[#tecUnitNumber].send.control.%X2 := #statDataExchangeSend.systemFixed.RunSequence;
   #interfaceHmi[#tecUnitNumber].send.control.%X3 := #statDataExchangeSend.systemFixed.DriveToHomePos;
   #interfaceHmi[#tecUnitNumber].send.control.%X4 := #statDataExchangeSend.systemFixed.DriveToRefPos;
   #interfaceHmi[#tecUnitNumber].send.control.%X5 := #statDataExchangeSend.systemFixed.JogFW;
   #interfaceHmi[#tecUnitNumber].send.control.%X6 := #statDataExchangeSend.systemFixed.JogBW;
   #interfaceHmi[#tecUnitNumber].send.control.%X7 := #statDataExchangeSend.systemFixed.ContinueFromWait;
   #interfaceHmi[#tecUnitNumber].send.control.%X8 := #statDataExchangeSend.systemFixed.strobe;
   #interfaceHmi[#tecUnitNumber].send.control.%X9 := #statDataExchangeSend.systemFixed.AckAdmin;
   #interfaceHmi[#tecUnitNumber].send.mpNum := #statDataExchangeSend.systemFixed.MP;
   #interfaceHmi[#tecUnitNumber].send.cfgMpNum := #statDataExchangeSend.systemFixed.Cfg_MP;
   #interfaceHmi[#tecUnitNumber].send.cfgAddress := #statDataExchangeSend.systemFixed.CFG_ADR;
   #interfaceHmi[#tecUnitNumber].send.cfgLength := #statDataExchangeSend.systemFixed.CFG_Length;
   #interfaceHmi[#tecUnitNumber].send.selectPage := #statDataExchangeSend.systemFixed.SelectedPage;
   #interfaceHmi[#tecUnitNumber].send.selectSeqeunce := #statDataExchangeSend.systemFixed.SelectSequence;
   #interfaceHmi[#tecUnitNumber].send.serverJogSpeed := #interfaceHmi[#tecUnitNumber].serverJogSpeedSet;
   #interfaceHmi[#tecUnitNumber].send.serverJogMaxForce := #interfaceHmi[#tecUnitNumber].serverJogMaxForceSet;
END_REGION

REGION Network 51: Generate Alarm for Pro Diag
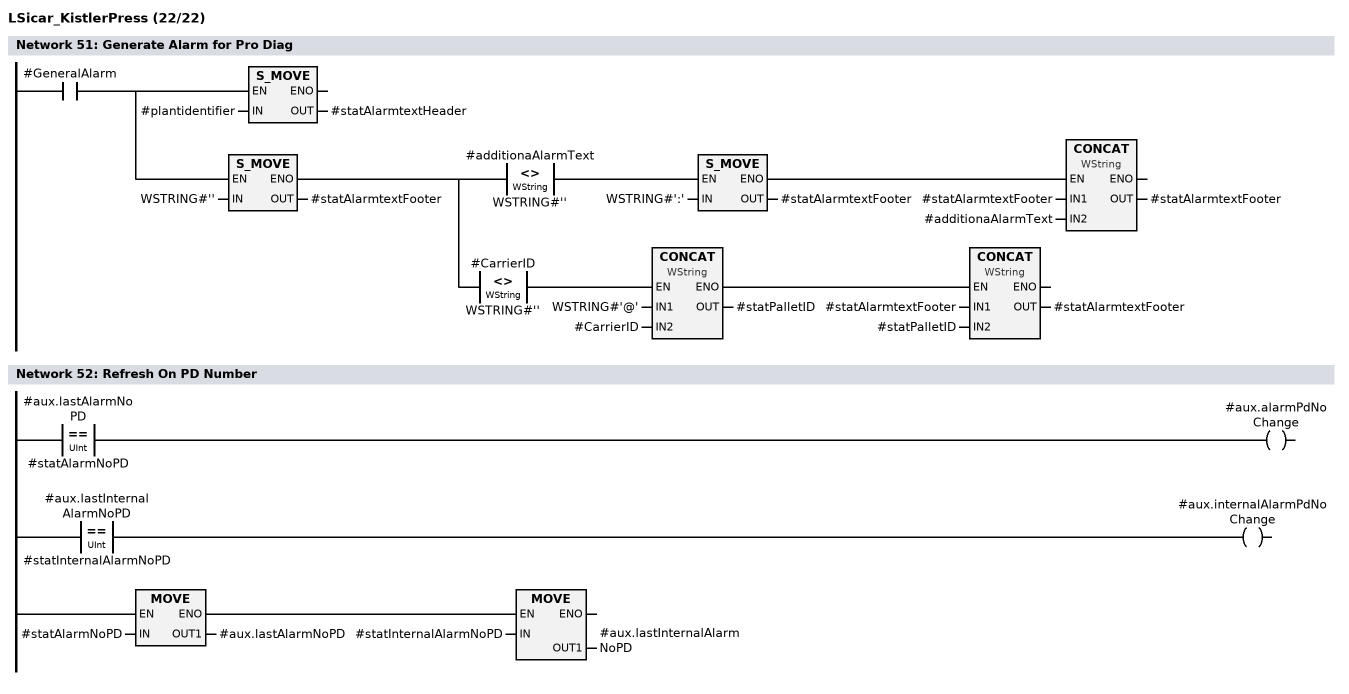
   RUNG wire#powerrail
      Contact( #GeneralAlarm )
      wire#w1
      S_Move(in := #plantidentifier, out => #statAlarmtextHeader)
   END_RUNG
   RUNG wire#w1
      S_Move(in := WSTRING#'', out => #statAlarmtextFooter)
      wire#w2
      { S7_Templates := "SrcType := WString" } NE_Contact(in1 := #additionaAlarmText, in2 := WSTRING#'')
      S_Move(in := WSTRING#':', out => #statAlarmtextFooter)
      { S7_Templates := "[card := 2, str_type := WString]" } CONCAT(IN1 := #statAlarmtextFooter, IN2 := #additionaAlarmText, OUT => #statAlarmtextFooter)
   END_RUNG
   RUNG wire#w2
      { S7_Templates := "SrcType := WString" } NE_Contact(in1 := #CarrierID, in2 := WSTRING#'')
      { S7_Templates := "[card := 2, str_type := WString]" } CONCAT(IN1 := WSTRING#'@', IN2 := #CarrierID, OUT => #statPalletID)
      { S7_Templates := "[card := 2, str_type := WString]" } CONCAT(IN1 := #statAlarmtextFooter, IN2 := #statPalletID, OUT => #statAlarmtextFooter)
   END_RUNG
   // the same network as SCL:
   IF #GeneralAlarm THEN
       #statAlarmtextHeader := #plantidentifier;
       #statAlarmtextFooter := WSTRING#'';
   END_IF;
   IF #GeneralAlarm AND (#additionaAlarmText <> WSTRING#'') THEN
       #statAlarmtextFooter := WSTRING#':';
       CONCAT(IN1 := #statAlarmtextFooter, IN2 := #additionaAlarmText, OUT => #statAlarmtextFooter);
   END_IF;
   CONCAT(EN := #GeneralAlarm AND (#CarrierID <> WSTRING#''),
          IN1 := WSTRING#'@',
          IN2 := #CarrierID,
          OUT => #statPalletID,
          ENO => #_w1);
   IF #_w1 THEN
       CONCAT(IN1 := #statAlarmtextFooter, IN2 := #statPalletID, OUT => #statAlarmtextFooter);
   END_IF;
END_REGION

REGION Network 52: Refresh On PD Number
   RUNG wire#powerrail
      { S7_Templates := "SrcType := UInt" } EQ_Contact(in1 := #aux.lastAlarmNoPD, in2 := #statAlarmNoPD)
      Coil( #aux.alarmPdNoChange )
   END_RUNG
   RUNG wire#powerrail
      { S7_Templates := "SrcType := UInt" } EQ_Contact(in1 := #aux.lastInternalAlarmNoPD, in2 := #statInternalAlarmNoPD)
      Coil( #aux.internalAlarmPdNoChange )
   END_RUNG
   RUNG wire#powerrail
      Move(in := #statAlarmNoPD, out1 => #aux.lastAlarmNoPD)
      Move(in := #statInternalAlarmNoPD, out1 => #aux.lastInternalAlarmNoPD)
   END_RUNG
   // the same network as SCL:
   #aux.alarmPdNoChange := #aux.lastAlarmNoPD = #statAlarmNoPD;
   #aux.internalAlarmPdNoChange := #aux.lastInternalAlarmNoPD = #statInternalAlarmNoPD;
   #aux.lastAlarmNoPD := #statAlarmNoPD;
   #aux.lastInternalAlarmNoPD := #statInternalAlarmNoPD;
END_REGION
END_FUNCTION_BLOCK
